(* Logix 5000 project; controller HP_SSC01hv vendor 1 type 14 code 158 rev 32.11; software revision 32.03; part 13 of 15 *)
(* tags used below, declared in another part *)
   A_C1_0200 : ALIAS FOR S_C1_FaultSafety.0;
   A_C1_0201 : ALIAS FOR S_C1_FaultSafety.1;
   A_C1_0202 : ALIAS FOR S_C1_FaultSafety.2;
   A_C1_0203 : ALIAS FOR S_C1_FaultSafety.3;
   A_C1_0204 : ALIAS FOR S_C1_FaultSafety.4;
   A_C1_0206 : ALIAS FOR S_C1_FaultSafety.6;
   A_C1_0208 : ALIAS FOR S_C1_FaultSafety.8;
   A_C1_0209 : ALIAS FOR S_C1_FaultSafety.9;
   A_C1_0210 : ALIAS FOR S_C1_FaultSafety.10;
   A_C1_0211 : ALIAS FOR S_C1_FaultSafety.11;
   A_C1_0216 : ALIAS FOR S_C1_FaultSafety.16;
   A_C1_0217 : ALIAS FOR S_C1_FaultSafety.17;
   A_C1_0220 : ALIAS FOR S_C1_FaultSafety.20;
   A_C2_0200 : ALIAS FOR S_C2_FaultSafety.0;
   A_C2_0201 : ALIAS FOR S_C2_FaultSafety.1;
   A_C2_0202 : ALIAS FOR S_C2_FaultSafety.2;
   A_C2_0203 : ALIAS FOR S_C2_FaultSafety.3;
   A_C2_0204 : ALIAS FOR S_C2_FaultSafety.4;
   A_C2_0206 : ALIAS FOR S_C2_FaultSafety.6;
   A_C2_0208 : ALIAS FOR S_C2_FaultSafety.8;
   A_C2_0209 : ALIAS FOR S_C2_FaultSafety.9;
   A_C2_0210 : ALIAS FOR S_C2_FaultSafety.10;
   A_C2_0211 : ALIAS FOR S_C2_FaultSafety.11;
   A_C2_0216 : ALIAS FOR S_C2_FaultSafety.16;
   A_C2_0217 : ALIAS FOR S_C2_FaultSafety.17;
   A_C2_0218 : ALIAS FOR S_C2_FaultSafety.18;
   A_C2_0219 : ALIAS FOR S_C2_FaultSafety.19;
   A_C2_0220 : ALIAS FOR S_C2_FaultSafety.20;
   A_C2_0221 : ALIAS FOR S_C2_FaultSafety.21;
   A_C2_0222 : ALIAS FOR S_C2_FaultSafety.22;
   A_C2_0223 : ALIAS FOR S_C2_FaultSafety.23;
   A_C2_0224 : ALIAS FOR S_C2_FaultSafety.24;
   A_C2_0230 : ALIAS FOR S_C2_FaultSafety.30;
   A_C2_0231 : ALIAS FOR S_C2_FaultSafety.31;
   A_S01_0104 : ALIAS FOR System_FaultSafeIO.4;
   A_S01_0122 : ALIAS FOR System_FaultSafeIO.22;
   C02_SafeMemory : Udt_Carsl_SafeData;
   C1_EvacInPositionTest : DINT;
   Multiplier : DINT;
   none : BOOL;
   RCS_CMD_EvacToStation : BOOL;
   RCS_SafeMemory_S01 : Udt_RCS_SafeData;
   RCS_SyncMotionEnable : BOOL;
   S1_C1_SafeOffFdbkRIN : REDUNDANT_INPUT;
   S_C1_AtEvacSpeed : BOOL;
   S_C1_BrakeTest : BOOL;
   S_C1_CircuitReset : BOOL;
   S_C1_CircuitReset_Pulse : TIMER;
   S_C1_DrawBridge_LS1 : ALIAS FOR SSC01_Safe2:I.Pt00Data;
   S_C1_DrawBridge_LS2 : ALIAS FOR SSC01_Safe2:I.Pt01Data;
   S_C1_DrawbridgeInputOK : BOOL;
   S_C1_DrawbridgeRIN : REDUNDANT_INPUT;
   S_C1_DumpTest : BOOL;
   S_C1_EvacOk : BOOL;
   S_C1_ExecuteInputOK : BOOL;
   S_C1_ExecutePB : BOOL;
   S_C1_FaultReset : BOOL;
   S_C1_FaultSafety : DINT;
   S_C1_FaultSafety_OK : BOOL;
   S_C1_FaultStandard : DINT;
   S_C1_FaultStandard_OK : BOOL;
   S_C1_FW_LocalOK : BOOL;
   S_C1_InEvacPosition : BOOL;
   S_C1_MaintEnable : BOOL;
   S_C1_MCC1_LIM_MCR : ALIAS FOR C1_Safe:O.Pt04Data;
   S_C1_ModeLocal : BOOL;
   S_C1_ModeRemote : BOOL;
   S_C1_MotionEnabled : BOOL;
   S_C1_MOTN_EXEC_RIN : REDUNDANT_INPUT;
   S_C1_MOTN_EXEC_SS_A : ALIAS FOR C1_Safe:I.Pt02Data;
   S_C1_MOTN_EXEC_SS_B : ALIAS FOR C1_Safe:I.Pt03Data;
   S_C1_MotorActualPositionX1000 : DINT;
   S_C1_MotorActualPositionX1000MOD60 : DINT;
   S_C1_MotorAverageVelocityX1000 : DINT;
   S_C1_MStop : EMERGENCY_STOP;
   S_C1_MSTOP_A : ALIAS FOR C1_Safe:I.Pt06Data;
   S_C1_MSTOP_B : ALIAS FOR C1_Safe:I.Pt07Data;
   S_C1_MSTOP_InputOK : BOOL;
   S_C1_MSTOP_LT : ALIAS FOR C1_Safe:O.Pt02Data;
   S_C1_NearOnPath : BOOL;
   S_C1_NearOnPathHi : DINT;
   S_C1_NearOnPathHiBase : DINT;
   S_C1_NearOnPathLow : DINT;
   S_C1_NearOnPathLowBase : DINT;
   S_C1_OffPath : BOOL;
   S_C1_OIT_FaultReset : BOOL;
   S_C1_OnPath : BOOL;
   S_C1_OnPathHi : DINT;
   S_C1_OnPathLow : DINT;
   S_C1_ONS : DINT;
   S_C1_ONS_CircuitFault : BOOL;
   S_C1_ONS_Status : BOOL;
   S_C1_OutputEnable : BOOL;
   S_C1_PathError : DINT;
   S_C1_PathErrorTest : DINT;
   S_C1_PathErrorTestTemp : DINT;
   S_C1_PathErrorTestTemp2 : DINT;
   S_C1_PathOffset : DINT;
   S_C1_PressureOK : ALIAS FOR C1_Safe:I.Pt05Data;
   S_C1_ResetTOF : TIMER;
   S_C1_SAFE_FDBK_Aux1 : BOOL;
   S_C1_SAFE_FDBK_Aux2 : BOOL;
   S_C1_SAFE_OFF_FDBK1 : ALIAS FOR C1_Safe:I.Pt01Data;
   S_C1_SAFE_OFF_FDBK2 : ALIAS FOR C1_Safe:I.Pt00Data;
   S_C1_SafeOff_ROUT : REDUNDANT_OUTPUT;
   S_C1_SafeOffEnabled : BOOL;
   S_C1_SafeOffEngaged : BOOL;
   S_C1_SafeOffInputOK : BOOL;
   S_C1_SAFETY_ENABLE_1 : ALIAS FOR C1_Safe:O.Pt00Data;
   S_C1_SAFETY_ENABLE_2 : ALIAS FOR C1_Safe:O.Pt01Data;
   S_C1_SS_RemoteMode : BOOL;
   S_C1_Stop0_OK : BOOL;
   S_C1_Stop1_OK : BOOL;
   S_C1_Stop1_OK_TOF : TIMER;
   S_C1_WindowAdderTemp1 : DINT;
   S_C1_WindowAdderTemp2 : DINT;
   S_C1_WindowAdderTemp3 : DINT;
   S_C2_AtEvacSpeed : BOOL;
   S_C2_BrakeRelease : ALIAS FOR C2_Safe:O.Pt06Data;
   S_C2_BrakeReleaseSelected : BOOL;
   S_C2_BrakeTest : BOOL;
   S_C2_CircuitReset : BOOL;
   S_C2_DrawbridgeInputOK : BOOL;
   S_C2_DrawbridgeRIN : REDUNDANT_INPUT;
   S_C2_DumpValveRelease : ALIAS FOR C2_Safe:O.Pt05Data;
   S_C2_DumpValveReleaseSelected : BOOL;
   S_C2_EncoderBuffer : DINT[4];
   S_C2_EncoderChange : DINT;
   S_C2_EncoderCounter : DINT;
   S_C2_EncoderCounts : DINT;
   S_C2_EncoderPositionAtHome : DINT;
   S_C2_EncoderPositionAtHomeSet : BOOL;
   S_C2_EncoderPositionDegree : DINT;
   S_C2_EncoderRev : DINT;
   S_C2_EncoderRevX1000 : DINT;
   S_C2_EncoderTemp : DINT;
   S_C2_EncoderTemp2 : DINT;
   S_C2_EvacOK : BOOL;
   S_C2_ExecuteInputOK : BOOL;
   S_C2_FaultReset : BOOL;
   S_C2_FaultSafety : DINT;
   S_C2_FaultSafety_OK : BOOL;
   S_C2_FaultStandard_OK : BOOL;
   S_C2_FaultTimer : TIMER[8];
   S_C2_Homed : BOOL;
   S_C2_HomeInputStatus : BOOL;
   S_C2_HomeSafePE : ALIAS FOR C2_Safe:I.Pt04Data;
   S_C2_InEvacPosition : BOOL;
   S_C2_ModeLocal : BOOL;
   S_C2_ModeRemote : BOOL;
   S_C2_MotorActualPositionX1000 : DINT;
   S_C2_MotorActualPositionX1000MOD60 : DINT;
   S_C2_MotorAverageVelocityX1000 : DINT;
   S_C2_MotorToEncoderError : DINT;
   S_C2_MStop : EMERGENCY_STOP;
   S_C2_MSTOP_InputOK : BOOL;
   S_C2_NearOnPath : BOOL;
   S_C2_NearOnPathHi : DINT;
   S_C2_NearOnPathHiBase : DINT;
   S_C2_NearOnPathLow : DINT;
   S_C2_NearOnPathLowBase : DINT;
   S_C2_OffPath : BOOL;
   S_C2_OnPath : BOOL;
   S_C2_OnPathHi : DINT;
   S_C2_OnPathLow : DINT;
   S_C2_ONS_Fault : BOOL;
   S_C2_OutputEnable : BOOL;
   S_C2_PathError : DINT;
   S_C2_PathErrorTest : DINT;
   S_C2_PathErrorTestTemp : DINT;
   S_C2_PathErrorTestTemp2 : DINT;
   S_C2_PathOffset : DINT;
   S_C2_PressureOK : ALIAS FOR C2_Safe:I.Pt05Data;
   S_C2_RemoteBrakeAndHomeSequence : DINT;
   S_C2_ReverseMotionDebounce : TIMER;
   S_C2_SAFE_OFF_FDBK1 : ALIAS FOR C2_Safe:I.Pt01Data;
   S_C2_SAFE_OFF_FDBK2 : ALIAS FOR C2_Safe:I.Pt00Data;
   S_C2_SafeOff_ROUT : REDUNDANT_OUTPUT;
   S_C2_SafeOffInputOK : BOOL;
   S_C2_SetEncoderHomePosition : BOOL;
   S_C2_WindowAdderTemp1 : DINT;
   S_C2_WindowAdderTemp2 : DINT;
   S_C2_WindowAdderTemp3 : DINT;
   S_EncoderRollover : DINT;
   S_EvacToStationTON : TIMER;
   S_FlashOn : TIMER;
   S_RCS_CMD_FaultReset : BOOL;
   S_RCS_EvacSpeedStart_TON : TIMER;
   S_RCS_MasterPositionDegrees : DINT;
   S_RCS_MotionEnable : BOOL;
   S_System_FaultStandard : DINT;
   SSC_Rail_BypassOK : BOOL;
   SSC_SafeFlt_OK : BOOL;
   SSC_SafetyIO_OK : BOOL;
   SSC_StdFlt_OK : BOOL;
   SSC_Stop0_OK : BOOL;
   SSC_Stop1_OK : BOOL;
(* SafeCarousel1, continued *)

ROUTINE SC125_PathError   (* ladder *)
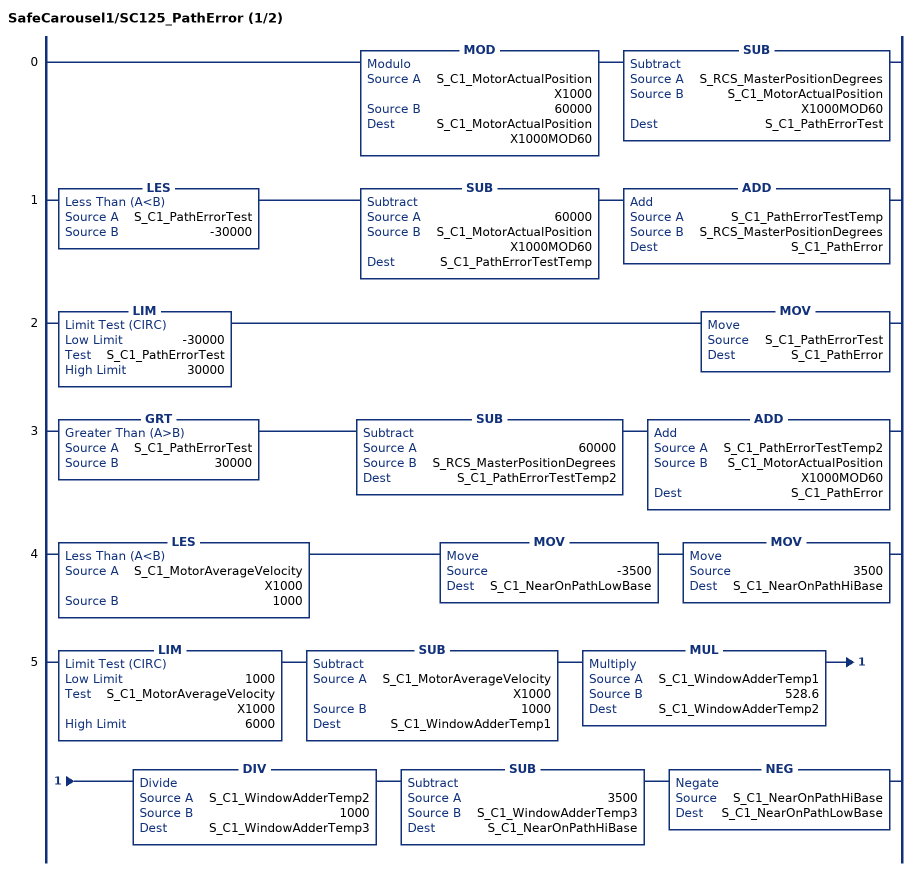
   0: MOD(S_C1_MotorActualPositionX1000,60000,S_C1_MotorActualPositionX1000MOD60)SUB(S_RCS_MasterPositionDegrees,S_C1_MotorActualPositionX1000MOD60,S_C1_PathErrorTest);
   1: LES(S_C1_PathErrorTest,-30000)SUB(60000,S_C1_MotorActualPositionX1000MOD60,S_C1_PathErrorTestTemp)ADD(S_C1_PathErrorTestTemp,S_RCS_MasterPositionDegrees,S_C1_PathError);
   2: LIM(-30000,S_C1_PathErrorTest,30000)MOV(S_C1_PathErrorTest,S_C1_PathError);
   3: GRT(S_C1_PathErrorTest,30000)SUB(60000,S_RCS_MasterPositionDegrees,S_C1_PathErrorTestTemp2)ADD(S_C1_PathErrorTestTemp2,S_C1_MotorActualPositionX1000MOD60,S_C1_PathError);
   4: LES(S_C1_MotorAverageVelocityX1000,1000)MOV(-3500,S_C1_NearOnPathLowBase)MOV(3500,S_C1_NearOnPathHiBase);
   5: LIM(1000,S_C1_MotorAverageVelocityX1000,6000)SUB(S_C1_MotorAverageVelocityX1000,1000,S_C1_WindowAdderTemp1)MUL(S_C1_WindowAdderTemp1,528.6,S_C1_WindowAdderTemp2)DIV(S_C1_WindowAdderTemp2,1000,S_C1_WindowAdderTemp3)SUB(3500,S_C1_WindowAdderTemp3,S_C1_NearOnPathHiBase)NEG(S_C1_NearOnPathHiBase,S_C1_NearOnPathLowBase);
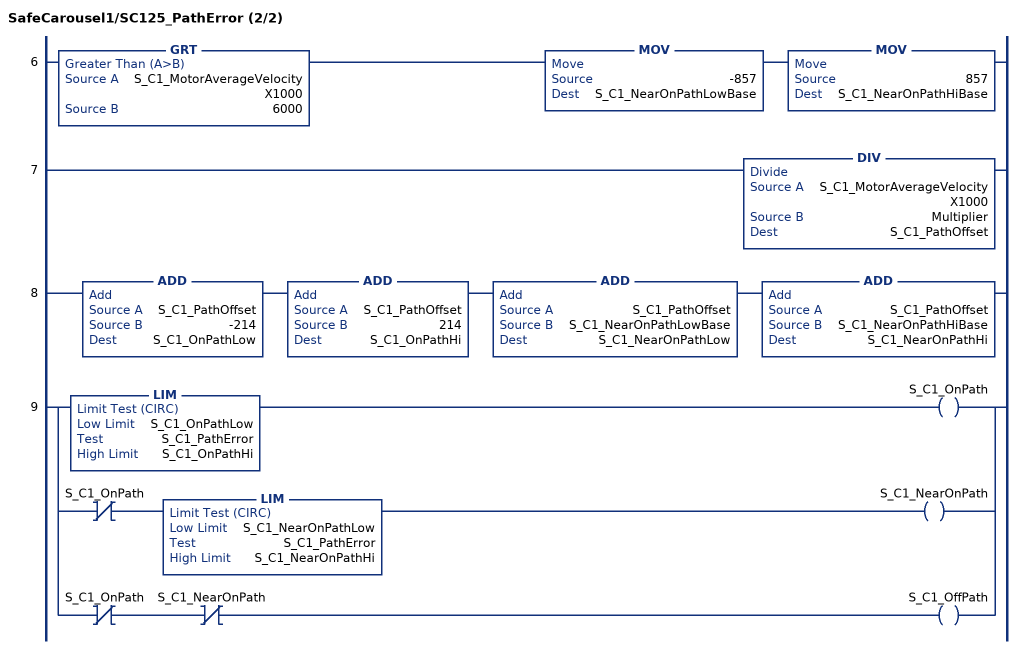
   6: GRT(S_C1_MotorAverageVelocityX1000,6000)MOV(-857,S_C1_NearOnPathLowBase)MOV(857,S_C1_NearOnPathHiBase);
   7: DIV(S_C1_MotorAverageVelocityX1000,Multiplier,S_C1_PathOffset);
   8: ADD(S_C1_PathOffset,-214,S_C1_OnPathLow)ADD(S_C1_PathOffset,214,S_C1_OnPathHi)ADD(S_C1_PathOffset,S_C1_NearOnPathLowBase,S_C1_NearOnPathLow)ADD(S_C1_PathOffset,S_C1_NearOnPathHiBase,S_C1_NearOnPathHi);
   9: [LIM(S_C1_OnPathLow,S_C1_PathError,S_C1_OnPathHi) OTE(S_C1_OnPath) ,XIO(S_C1_OnPath) LIM(S_C1_NearOnPathLow,S_C1_PathError,S_C1_NearOnPathHi) OTE(S_C1_NearOnPath) ,XIO(S_C1_OnPath) XIO(S_C1_NearOnPath) OTE(S_C1_OffPath) ];
END_ROUTINE

ROUTINE SC130_SafetyInputs   (* ladder *)
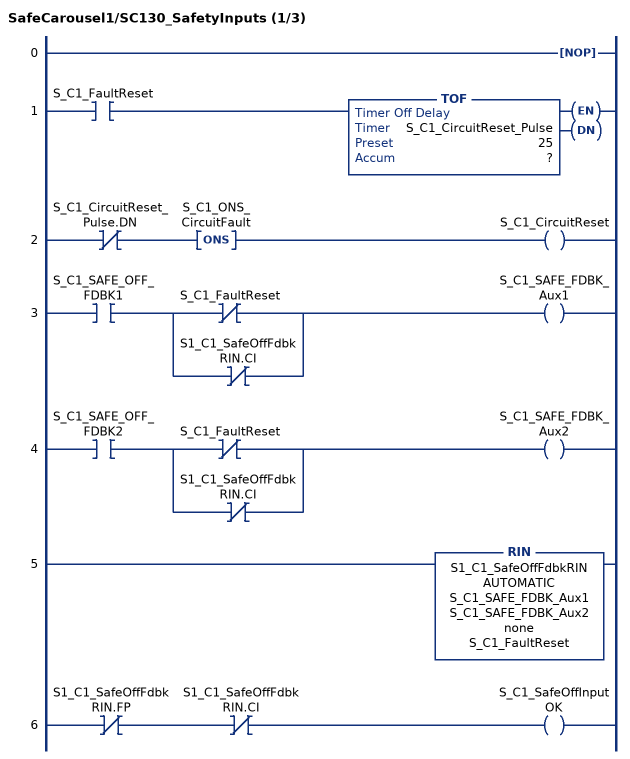
   0: NOP();
   1: XIC(S_C1_FaultReset)TOF(S_C1_CircuitReset_Pulse,?,?);
   2: XIO(S_C1_CircuitReset_Pulse.DN)ONS(S_C1_ONS_CircuitFault)OTE(S_C1_CircuitReset);
   3: XIC(S_C1_SAFE_OFF_FDBK1)[XIO(S_C1_FaultReset) ,XIO(S1_C1_SafeOffFdbkRIN.CI) ]OTE(S_C1_SAFE_FDBK_Aux1);
   4: XIC(S_C1_SAFE_OFF_FDBK2)[XIO(S_C1_FaultReset) ,XIO(S1_C1_SafeOffFdbkRIN.CI) ]OTE(S_C1_SAFE_FDBK_Aux2);
   5: RIN(S1_C1_SafeOffFdbkRIN,AUTOMATIC,S_C1_SAFE_FDBK_Aux1,S_C1_SAFE_FDBK_Aux2,none,S_C1_FaultReset);
   6: XIO(S1_C1_SafeOffFdbkRIN.FP)XIO(S1_C1_SafeOffFdbkRIN.CI)OTE(S_C1_SafeOffInputOK);
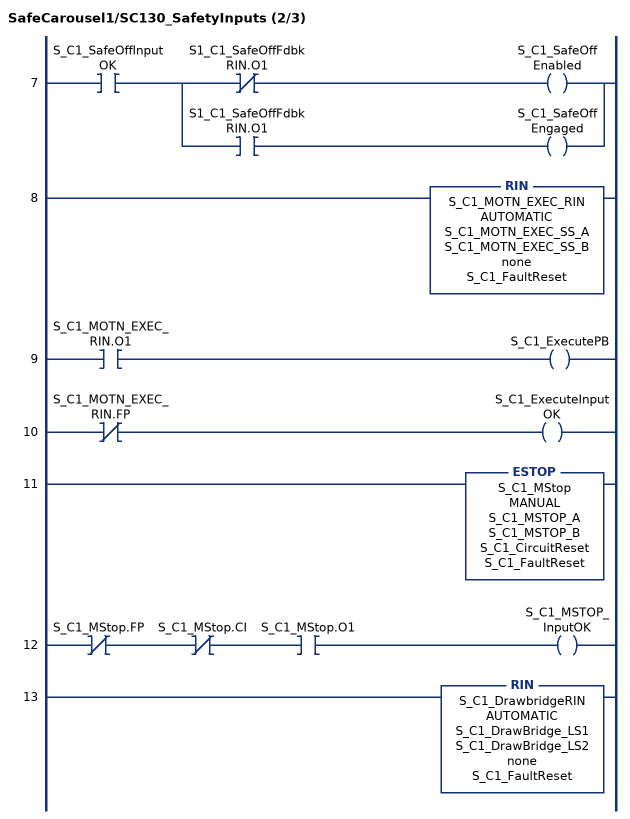
   7: XIC(S_C1_SafeOffInputOK)[XIO(S1_C1_SafeOffFdbkRIN.O1) OTE(S_C1_SafeOffEnabled) ,XIC(S1_C1_SafeOffFdbkRIN.O1) OTE(S_C1_SafeOffEngaged) ];
   8: RIN(S_C1_MOTN_EXEC_RIN,AUTOMATIC,S_C1_MOTN_EXEC_SS_A,S_C1_MOTN_EXEC_SS_B,none,S_C1_FaultReset);
   9: XIC(S_C1_MOTN_EXEC_RIN.O1)OTE(S_C1_ExecutePB);
   10: XIO(S_C1_MOTN_EXEC_RIN.FP)OTE(S_C1_ExecuteInputOK);
   11: ESTOP(S_C1_MStop,MANUAL,S_C1_MSTOP_A,S_C1_MSTOP_B,S_C1_CircuitReset,S_C1_FaultReset);
   12: XIO(S_C1_MStop.FP)XIO(S_C1_MStop.CI)XIC(S_C1_MStop.O1)OTE(S_C1_MSTOP_InputOK);
   13: RIN(S_C1_DrawbridgeRIN,AUTOMATIC,S_C1_DrawBridge_LS1,S_C1_DrawBridge_LS2,none,S_C1_FaultReset);
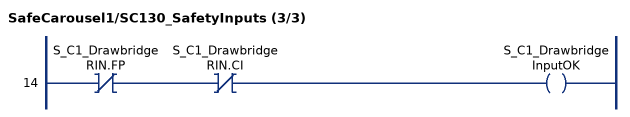
   14: XIO(S_C1_DrawbridgeRIN.FP)XIO(S_C1_DrawbridgeRIN.CI)OTE(S_C1_DrawbridgeInputOK);
END_ROUTINE

ROUTINE SC135_SafetyOutputs   (* ladder *)
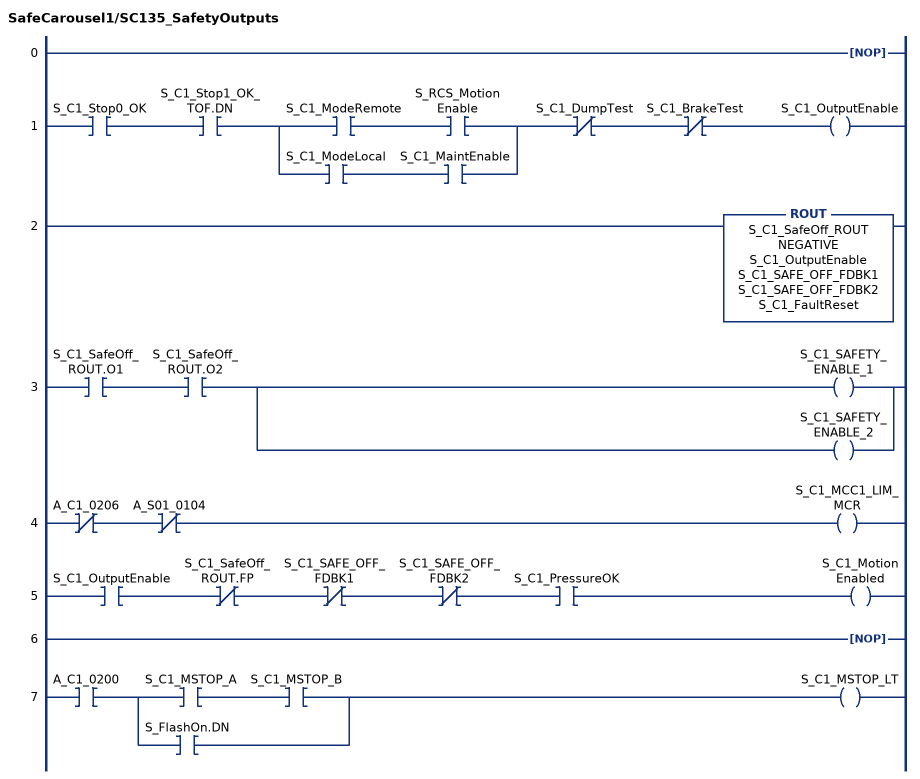
   0: NOP();
   1: XIC(S_C1_Stop0_OK)XIC(S_C1_Stop1_OK_TOF.DN)[XIC(S_C1_ModeRemote) XIC(S_RCS_MotionEnable) ,XIC(S_C1_ModeLocal) XIC(S_C1_MaintEnable) ]XIO(S_C1_DumpTest)XIO(S_C1_BrakeTest)OTE(S_C1_OutputEnable);
   2: ROUT(S_C1_SafeOff_ROUT,NEGATIVE,S_C1_OutputEnable,S_C1_SAFE_OFF_FDBK1,S_C1_SAFE_OFF_FDBK2,S_C1_FaultReset);
   3: XIC(S_C1_SafeOff_ROUT.O1)XIC(S_C1_SafeOff_ROUT.O2)[OTE(S_C1_SAFETY_ENABLE_1) ,OTE(S_C1_SAFETY_ENABLE_2) ];
   4: XIO(A_C1_0206)XIO(A_S01_0104)OTE(S_C1_MCC1_LIM_MCR);
   5: XIC(S_C1_OutputEnable)XIO(S_C1_SafeOff_ROUT.FP)XIO(S_C1_SAFE_OFF_FDBK1)XIO(S_C1_SAFE_OFF_FDBK2)XIC(S_C1_PressureOK)OTE(S_C1_MotionEnabled);
   6: NOP();
   7: XIC(A_C1_0200)[XIC(S_C1_MSTOP_A) XIC(S_C1_MSTOP_B) ,XIC(S_FlashOn.DN) ]OTE(S_C1_MSTOP_LT);
END_ROUTINE

ROUTINE SC140_Status   (* ladder *)
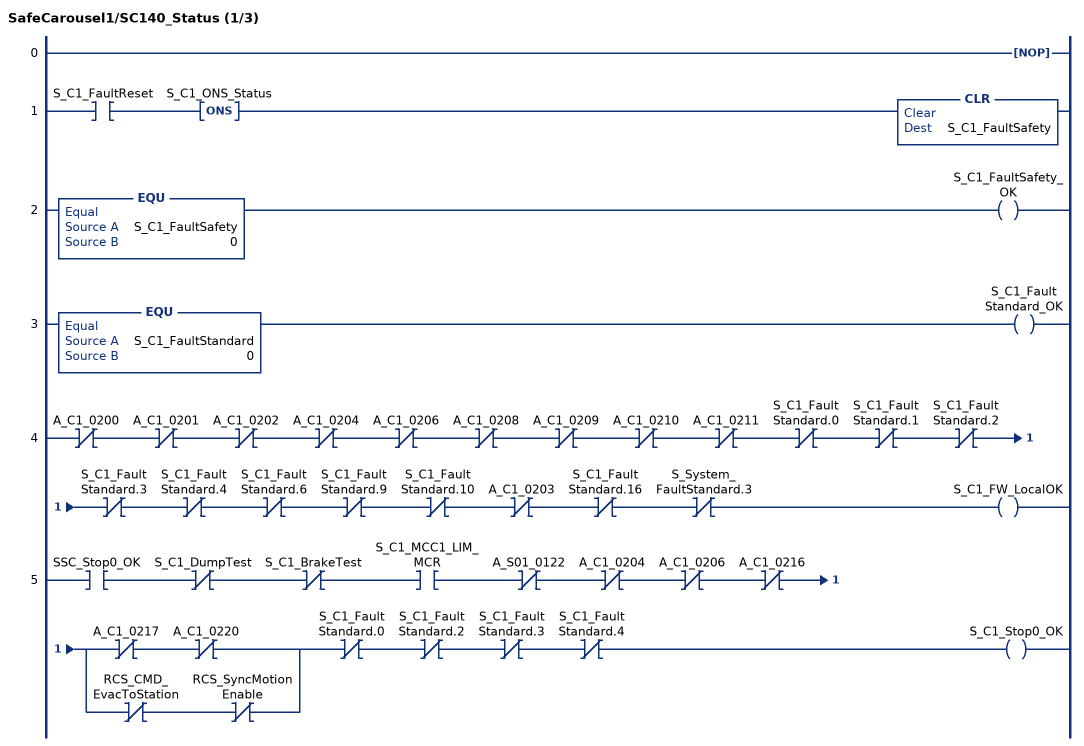
   0: NOP();
   1: XIC(S_C1_FaultReset)ONS(S_C1_ONS_Status)CLR(S_C1_FaultSafety);
   2: EQU(S_C1_FaultSafety,0)OTE(S_C1_FaultSafety_OK);
   3: EQU(S_C1_FaultStandard,0)OTE(S_C1_FaultStandard_OK);
   4: XIO(A_C1_0200)XIO(A_C1_0201)XIO(A_C1_0202)XIO(A_C1_0204)XIO(A_C1_0206)XIO(A_C1_0208)XIO(A_C1_0209)XIO(A_C1_0210)XIO(A_C1_0211)XIO(S_C1_FaultStandard.0)XIO(S_C1_FaultStandard.1)XIO(S_C1_FaultStandard.2)XIO(S_C1_FaultStandard.3)XIO(S_C1_FaultStandard.4)XIO(S_C1_FaultStandard.6)XIO(S_C1_FaultStandard.9)XIO(S_C1_FaultStandard.10)XIO(A_C1_0203)XIO(S_C1_FaultStandard.16)XIO(S_System_FaultStandard.3)OTE(S_C1_FW_LocalOK);
   5: XIC(SSC_Stop0_OK)XIO(S_C1_DumpTest)XIO(S_C1_BrakeTest)XIC(S_C1_MCC1_LIM_MCR)XIO(A_S01_0122)XIO(A_C1_0204)XIO(A_C1_0206)XIO(A_C1_0216)[XIO(A_C1_0217) XIO(A_C1_0220) ,XIO(RCS_CMD_EvacToStation) XIO(RCS_SyncMotionEnable) ]XIO(S_C1_FaultStandard.0)XIO(S_C1_FaultStandard.2)XIO(S_C1_FaultStandard.3)XIO(S_C1_FaultStandard.4)OTE(S_C1_Stop0_OK);
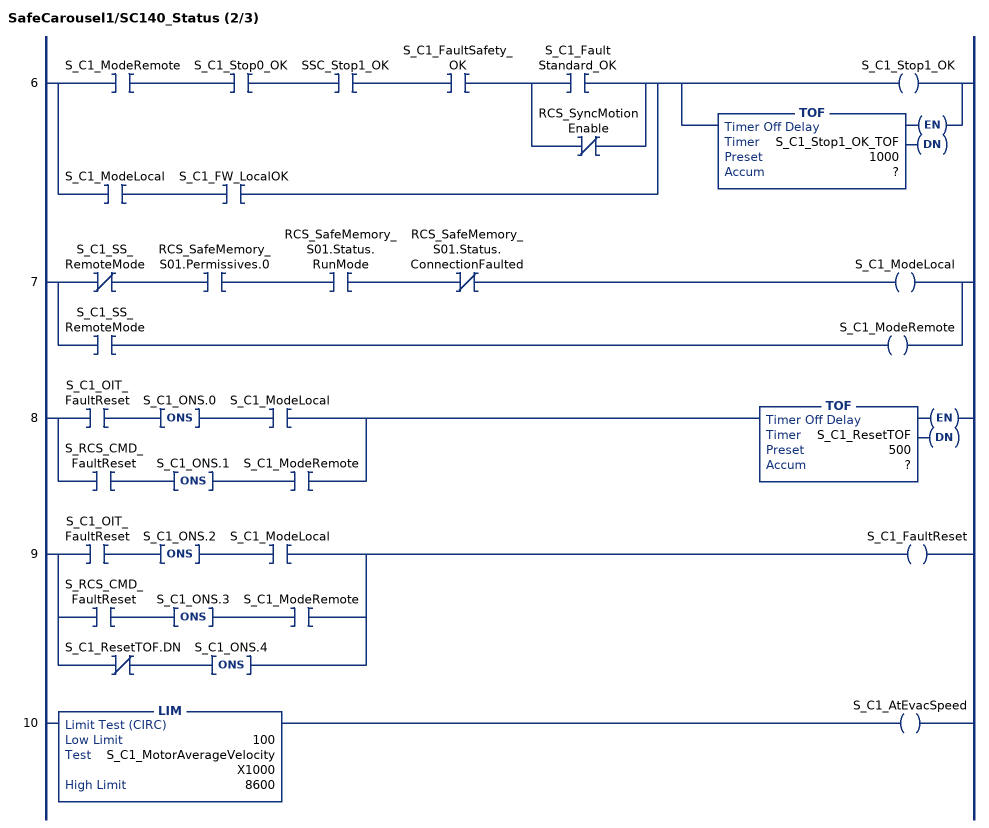
   6: [XIC(S_C1_ModeRemote) XIC(S_C1_Stop0_OK) XIC(SSC_Stop1_OK) XIC(S_C1_FaultSafety_OK) [XIC(S_C1_FaultStandard_OK) ,XIO(RCS_SyncMotionEnable) ] ,XIC(S_C1_ModeLocal) XIC(S_C1_FW_LocalOK) ][OTE(S_C1_Stop1_OK) ,TOF(S_C1_Stop1_OK_TOF,?,?) ];
   7: [XIO(S_C1_SS_RemoteMode) XIC(RCS_SafeMemory_S01.Permissives.0) XIC(RCS_SafeMemory_S01.Status.RunMode) XIO(RCS_SafeMemory_S01.Status.ConnectionFaulted) OTE(S_C1_ModeLocal) ,XIC(S_C1_SS_RemoteMode) OTE(S_C1_ModeRemote) ];
   8: [XIC(S_C1_OIT_FaultReset) ONS(S_C1_ONS.0) XIC(S_C1_ModeLocal) ,XIC(S_RCS_CMD_FaultReset) ONS(S_C1_ONS.1) XIC(S_C1_ModeRemote) ]TOF(S_C1_ResetTOF,?,?);
   9: [XIC(S_C1_OIT_FaultReset) ONS(S_C1_ONS.2) XIC(S_C1_ModeLocal) ,XIC(S_RCS_CMD_FaultReset) ONS(S_C1_ONS.3) XIC(S_C1_ModeRemote) ,XIO(S_C1_ResetTOF.DN) ONS(S_C1_ONS.4) ]OTE(S_C1_FaultReset);
   10: LIM(100,S_C1_MotorAverageVelocityX1000,8600)OTE(S_C1_AtEvacSpeed);
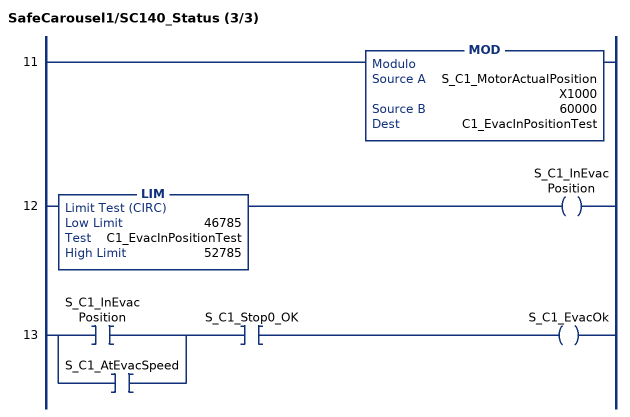
   11: MOD(S_C1_MotorActualPositionX1000,60000,C1_EvacInPositionTest);
   12: LIM(46785,C1_EvacInPositionTest,52785)OTE(S_C1_InEvacPosition);
   13: [XIC(S_C1_InEvacPosition) ,XIC(S_C1_AtEvacSpeed) ]XIC(S_C1_Stop0_OK)OTE(S_C1_EvacOk);
END_ROUTINE
END_PROGRAM

PROGRAM SafeCarousel2   (* main routine SC200_Main, safety *)

ROUTINE SC200_Main   (* ladder *)
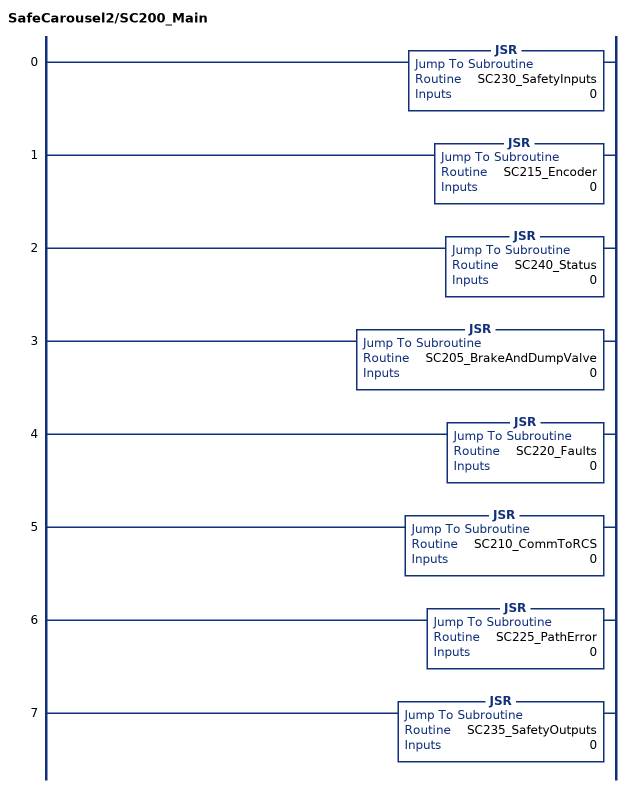
   0: JSR(SC230_SafetyInputs,0);
   1: JSR(SC215_Encoder,0);
   2: JSR(SC240_Status,0);
   3: JSR(SC205_BrakeAndDumpValve,0);
   4: JSR(SC220_Faults,0);
   5: JSR(SC210_CommToRCS,0);
   6: JSR(SC225_PathError,0);
   7: JSR(SC235_SafetyOutputs,0);
END_ROUTINE

ROUTINE SC205_BrakeAndDumpValve   (* ladder *)
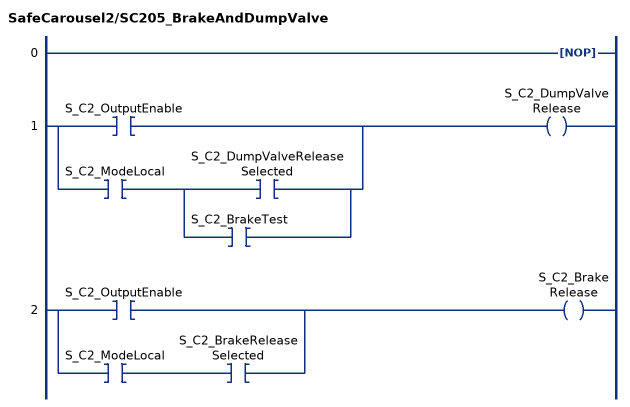
   0: NOP();
   1: [XIC(S_C2_OutputEnable) ,XIC(S_C2_ModeLocal) [XIC(S_C2_DumpValveReleaseSelected) ,XIC(S_C2_BrakeTest) ] ]OTE(S_C2_DumpValveRelease);
   2: [XIC(S_C2_OutputEnable) ,XIC(S_C2_ModeLocal) XIC(S_C2_BrakeReleaseSelected) ]OTE(S_C2_BrakeRelease);
END_ROUTINE

ROUTINE SC210_CommToRCS   (* ladder *)
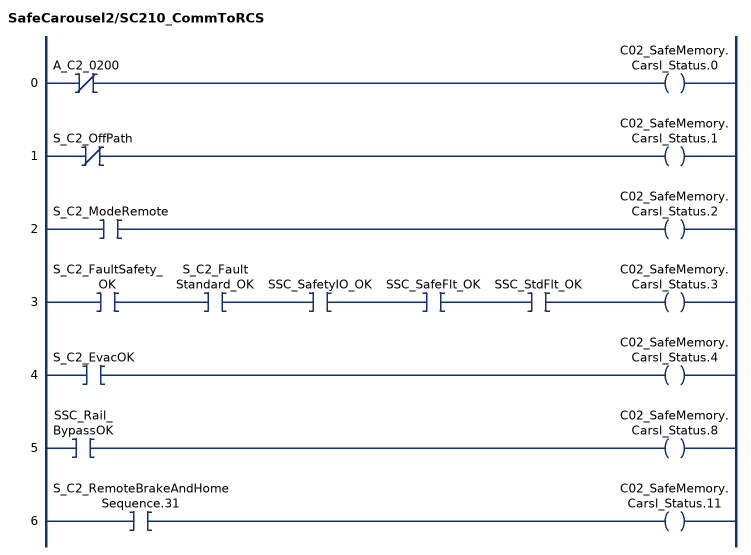
   0: XIO(A_C2_0200)OTE(C02_SafeMemory.Carsl_Status.0);
   1: XIO(S_C2_OffPath)OTE(C02_SafeMemory.Carsl_Status.1);
   2: XIC(S_C2_ModeRemote)OTE(C02_SafeMemory.Carsl_Status.2);
   3: XIC(S_C2_FaultSafety_OK)XIC(S_C2_FaultStandard_OK)XIC(SSC_SafetyIO_OK)XIC(SSC_SafeFlt_OK)XIC(SSC_StdFlt_OK)OTE(C02_SafeMemory.Carsl_Status.3);
   4: XIC(S_C2_EvacOK)OTE(C02_SafeMemory.Carsl_Status.4);
   5: XIC(SSC_Rail_BypassOK)OTE(C02_SafeMemory.Carsl_Status.8);
   6: XIC(S_C2_RemoteBrakeAndHomeSequence.31)OTE(C02_SafeMemory.Carsl_Status.11);
END_ROUTINE

ROUTINE SC215_Encoder   (* ladder *)
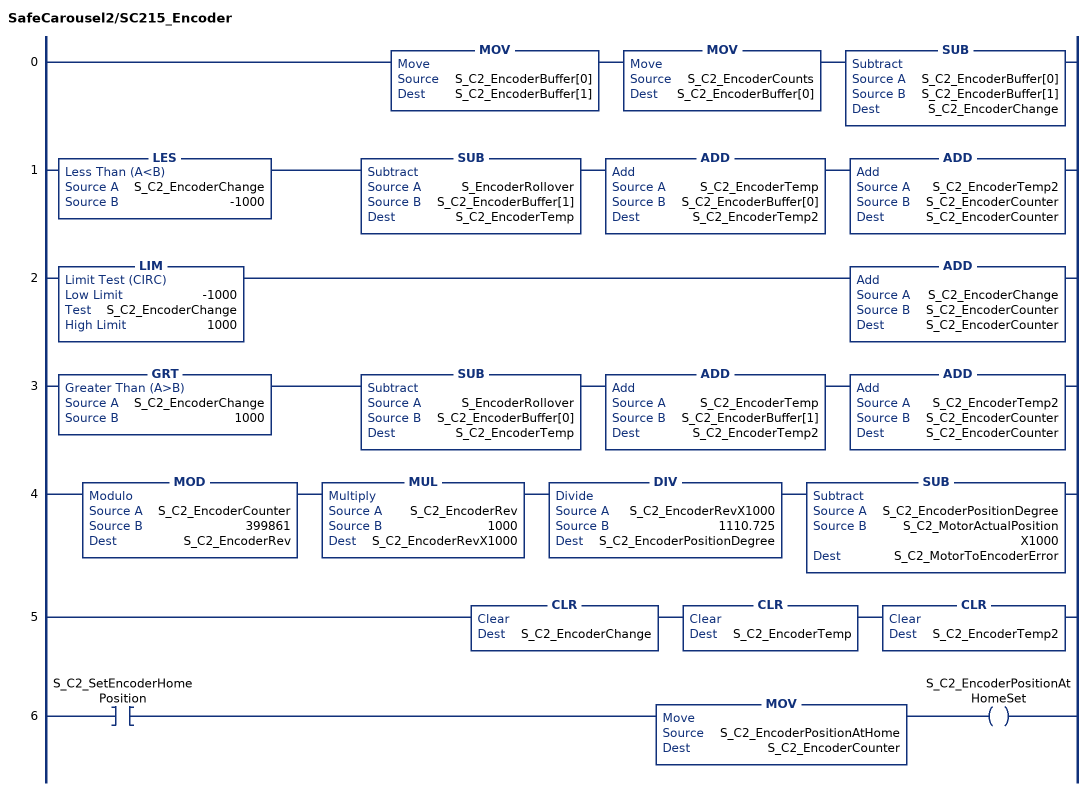
   0: MOV(S_C2_EncoderBuffer[0],S_C2_EncoderBuffer[1])MOV(S_C2_EncoderCounts,S_C2_EncoderBuffer[0])SUB(S_C2_EncoderBuffer[0],S_C2_EncoderBuffer[1],S_C2_EncoderChange);
   1: LES(S_C2_EncoderChange,-1000)SUB(S_EncoderRollover,S_C2_EncoderBuffer[1],S_C2_EncoderTemp)ADD(S_C2_EncoderTemp,S_C2_EncoderBuffer[0],S_C2_EncoderTemp2)ADD(S_C2_EncoderTemp2,S_C2_EncoderCounter,S_C2_EncoderCounter);
   2: LIM(-1000,S_C2_EncoderChange,1000)ADD(S_C2_EncoderChange,S_C2_EncoderCounter,S_C2_EncoderCounter);
   3: GRT(S_C2_EncoderChange,1000)SUB(S_EncoderRollover,S_C2_EncoderBuffer[0],S_C2_EncoderTemp)ADD(S_C2_EncoderTemp,S_C2_EncoderBuffer[1],S_C2_EncoderTemp2)ADD(S_C2_EncoderTemp2,S_C2_EncoderCounter,S_C2_EncoderCounter);
   4: MOD(S_C2_EncoderCounter,399861,S_C2_EncoderRev)MUL(S_C2_EncoderRev,1000,S_C2_EncoderRevX1000)DIV(S_C2_EncoderRevX1000,1110.725,S_C2_EncoderPositionDegree)SUB(S_C2_EncoderPositionDegree,S_C2_MotorActualPositionX1000,S_C2_MotorToEncoderError);
   5: CLR(S_C2_EncoderChange)CLR(S_C2_EncoderTemp)CLR(S_C2_EncoderTemp2);
   6: XIC(S_C2_SetEncoderHomePosition)MOV(S_C2_EncoderPositionAtHome,S_C2_EncoderCounter)OTE(S_C2_EncoderPositionAtHomeSet);
END_ROUTINE

ROUTINE SC220_Faults   (* ladder *)
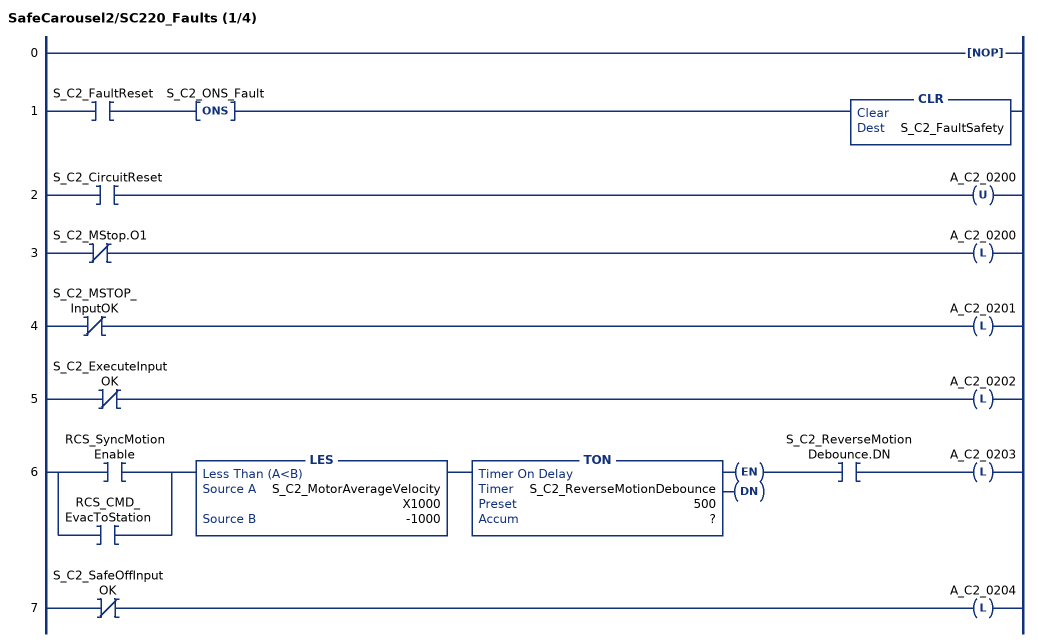
   0: NOP();
   1: XIC(S_C2_FaultReset)ONS(S_C2_ONS_Fault)CLR(S_C2_FaultSafety);
   2: XIC(S_C2_CircuitReset)OTU(A_C2_0200);
   3: XIO(S_C2_MStop.O1)OTL(A_C2_0200);
   4: XIO(S_C2_MSTOP_InputOK)OTL(A_C2_0201);
   5: XIO(S_C2_ExecuteInputOK)OTL(A_C2_0202);
   6: [XIC(RCS_SyncMotionEnable) ,XIC(RCS_CMD_EvacToStation) ]LES(S_C2_MotorAverageVelocityX1000,-1000)TON(S_C2_ReverseMotionDebounce,?,?)XIC(S_C2_ReverseMotionDebounce.DN)OTL(A_C2_0203);
   7: XIO(S_C2_SafeOffInputOK)OTL(A_C2_0204);
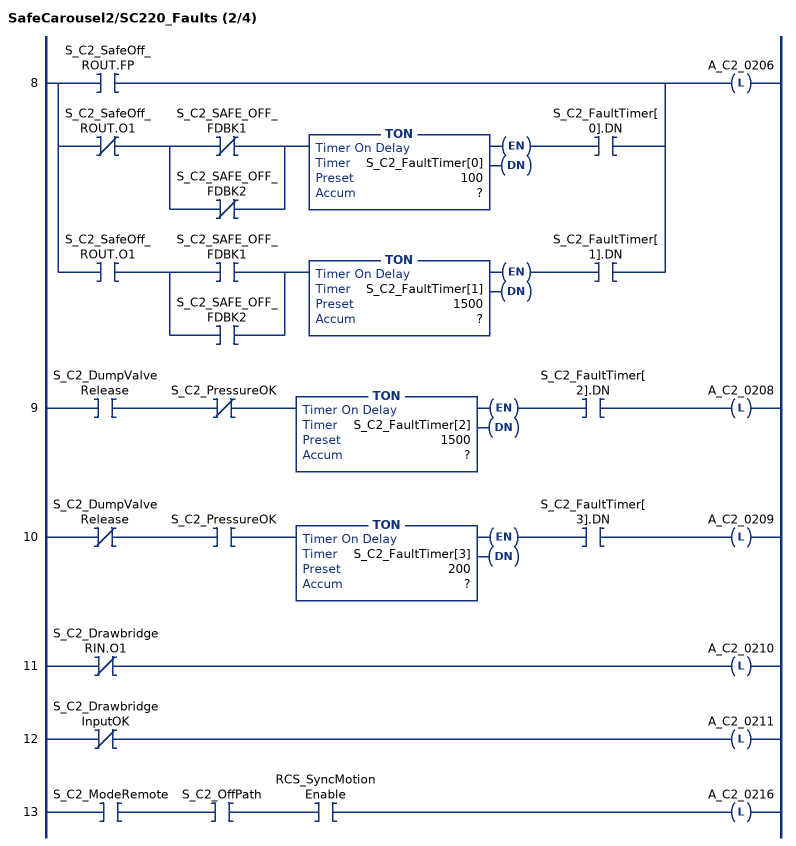
   8: [XIC(S_C2_SafeOff_ROUT.FP) ,XIO(S_C2_SafeOff_ROUT.O1) [XIO(S_C2_SAFE_OFF_FDBK1) ,XIO(S_C2_SAFE_OFF_FDBK2) ] TON(S_C2_FaultTimer[0],?,?) XIC(S_C2_FaultTimer[0].DN) ,XIC(S_C2_SafeOff_ROUT.O1) [XIC(S_C2_SAFE_OFF_FDBK1) ,XIC(S_C2_SAFE_OFF_FDBK2) ] TON(S_C2_FaultTimer[1],?,?) XIC(S_C2_FaultTimer[1].DN) ]OTL(A_C2_0206);
   9: XIC(S_C2_DumpValveRelease)XIO(S_C2_PressureOK)TON(S_C2_FaultTimer[2],?,?)XIC(S_C2_FaultTimer[2].DN)OTL(A_C2_0208);
   10: XIO(S_C2_DumpValveRelease)XIC(S_C2_PressureOK)TON(S_C2_FaultTimer[3],?,?)XIC(S_C2_FaultTimer[3].DN)OTL(A_C2_0209);
   11: XIO(S_C2_DrawbridgeRIN.O1)OTL(A_C2_0210);
   12: XIO(S_C2_DrawbridgeInputOK)OTL(A_C2_0211);
   13: XIC(S_C2_ModeRemote)XIC(S_C2_OffPath)XIC(RCS_SyncMotionEnable)OTL(A_C2_0216);
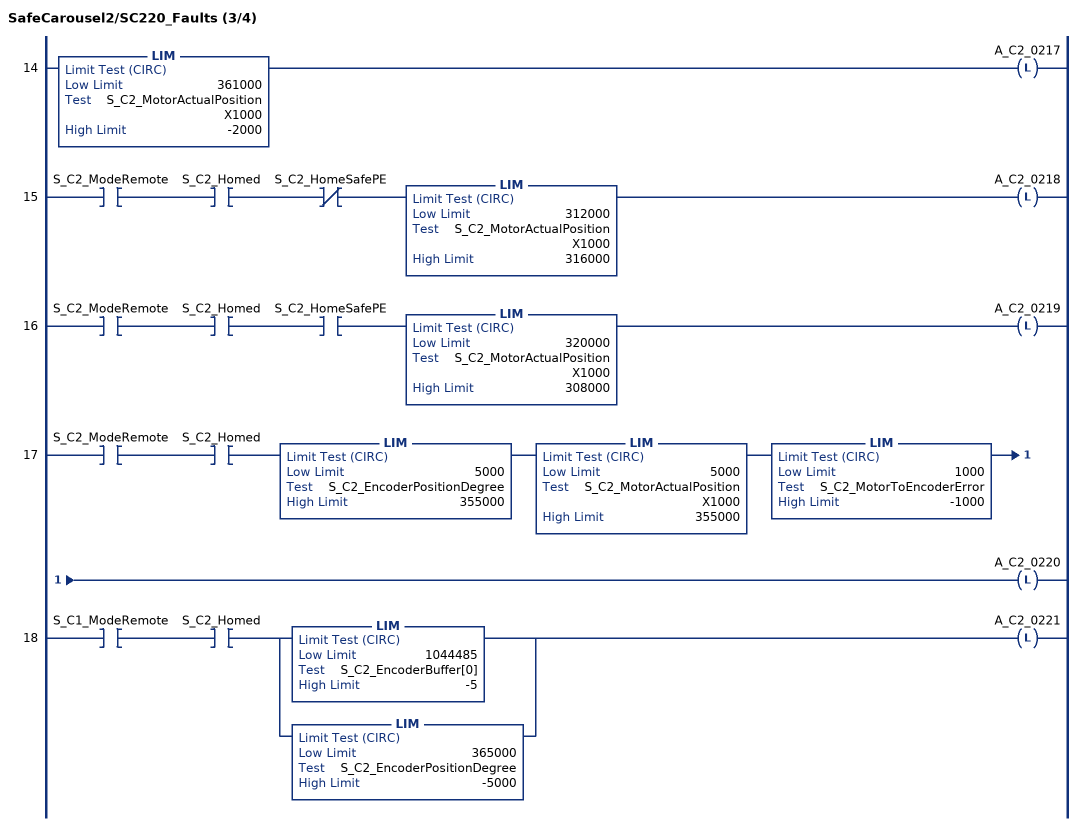
   14: LIM(361000,S_C2_MotorActualPositionX1000,-2000)OTL(A_C2_0217);
   15: XIC(S_C2_ModeRemote)XIC(S_C2_Homed)XIO(S_C2_HomeSafePE)LIM(312000,S_C2_MotorActualPositionX1000,316000)OTL(A_C2_0218);
   16: XIC(S_C2_ModeRemote)XIC(S_C2_Homed)XIC(S_C2_HomeSafePE)LIM(320000,S_C2_MotorActualPositionX1000,308000)OTL(A_C2_0219);
   17: XIC(S_C2_ModeRemote)XIC(S_C2_Homed)LIM(5000,S_C2_EncoderPositionDegree,355000)LIM(5000,S_C2_MotorActualPositionX1000,355000)LIM(1000,S_C2_MotorToEncoderError,-1000)OTL(A_C2_0220);
   18: XIC(S_C1_ModeRemote)XIC(S_C2_Homed)[LIM(1044485,S_C2_EncoderBuffer[0],-5) ,LIM(365000,S_C2_EncoderPositionDegree,-5000) ]OTL(A_C2_0221);
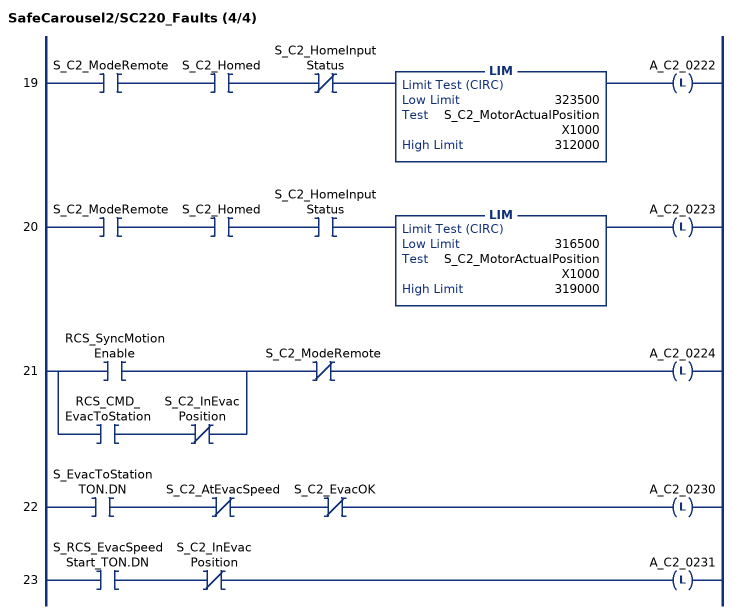
   19: XIC(S_C2_ModeRemote)XIC(S_C2_Homed)XIO(S_C2_HomeInputStatus)LIM(323500,S_C2_MotorActualPositionX1000,312000)OTL(A_C2_0222);
   20: XIC(S_C2_ModeRemote)XIC(S_C2_Homed)XIC(S_C2_HomeInputStatus)LIM(316500,S_C2_MotorActualPositionX1000,319000)OTL(A_C2_0223);
   21: [XIC(RCS_SyncMotionEnable) ,XIC(RCS_CMD_EvacToStation) XIO(S_C2_InEvacPosition) ]XIO(S_C2_ModeRemote)OTL(A_C2_0224);
   22: XIC(S_EvacToStationTON.DN)XIO(S_C2_AtEvacSpeed)XIO(S_C2_EvacOK)OTL(A_C2_0230);
   23: XIC(S_RCS_EvacSpeedStart_TON.DN)XIO(S_C2_InEvacPosition)OTL(A_C2_0231);
END_ROUTINE

ROUTINE SC225_PathError   (* ladder *)
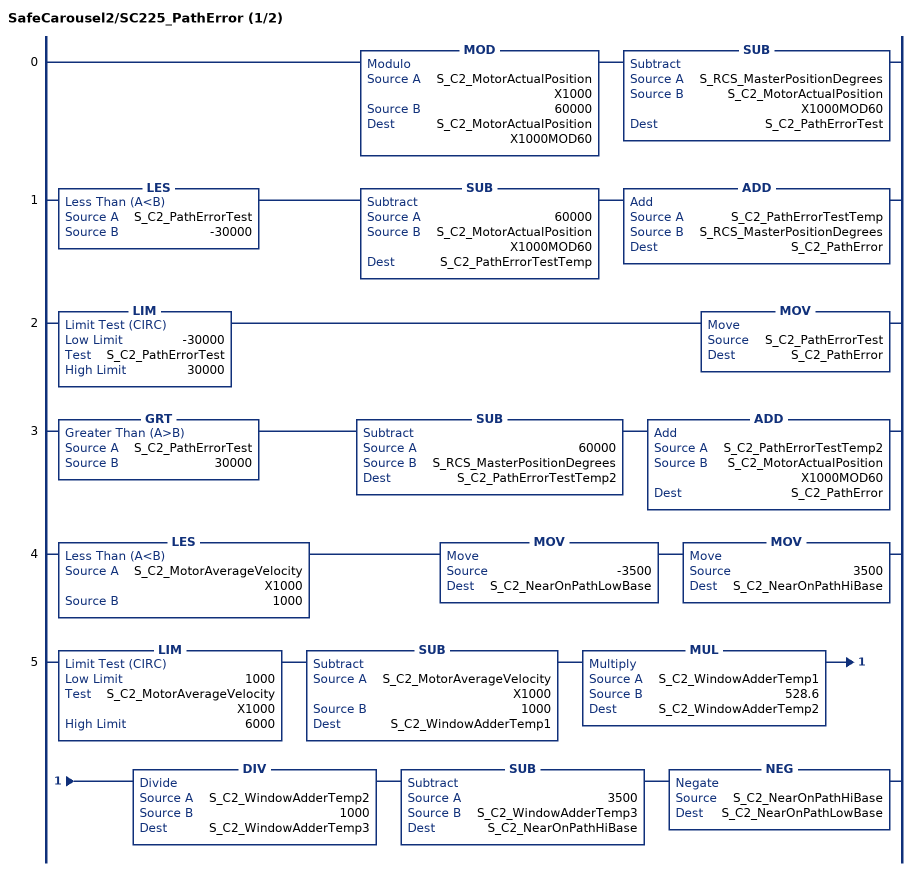
   0: MOD(S_C2_MotorActualPositionX1000,60000,S_C2_MotorActualPositionX1000MOD60)SUB(S_RCS_MasterPositionDegrees,S_C2_MotorActualPositionX1000MOD60,S_C2_PathErrorTest);
   1: LES(S_C2_PathErrorTest,-30000)SUB(60000,S_C2_MotorActualPositionX1000MOD60,S_C2_PathErrorTestTemp)ADD(S_C2_PathErrorTestTemp,S_RCS_MasterPositionDegrees,S_C2_PathError);
   2: LIM(-30000,S_C2_PathErrorTest,30000)MOV(S_C2_PathErrorTest,S_C2_PathError);
   3: GRT(S_C2_PathErrorTest,30000)SUB(60000,S_RCS_MasterPositionDegrees,S_C2_PathErrorTestTemp2)ADD(S_C2_PathErrorTestTemp2,S_C2_MotorActualPositionX1000MOD60,S_C2_PathError);
   4: LES(S_C2_MotorAverageVelocityX1000,1000)MOV(-3500,S_C2_NearOnPathLowBase)MOV(3500,S_C2_NearOnPathHiBase);
   5: LIM(1000,S_C2_MotorAverageVelocityX1000,6000)SUB(S_C2_MotorAverageVelocityX1000,1000,S_C2_WindowAdderTemp1)MUL(S_C2_WindowAdderTemp1,528.6,S_C2_WindowAdderTemp2)DIV(S_C2_WindowAdderTemp2,1000,S_C2_WindowAdderTemp3)SUB(3500,S_C2_WindowAdderTemp3,S_C2_NearOnPathHiBase)NEG(S_C2_NearOnPathHiBase,S_C2_NearOnPathLowBase);
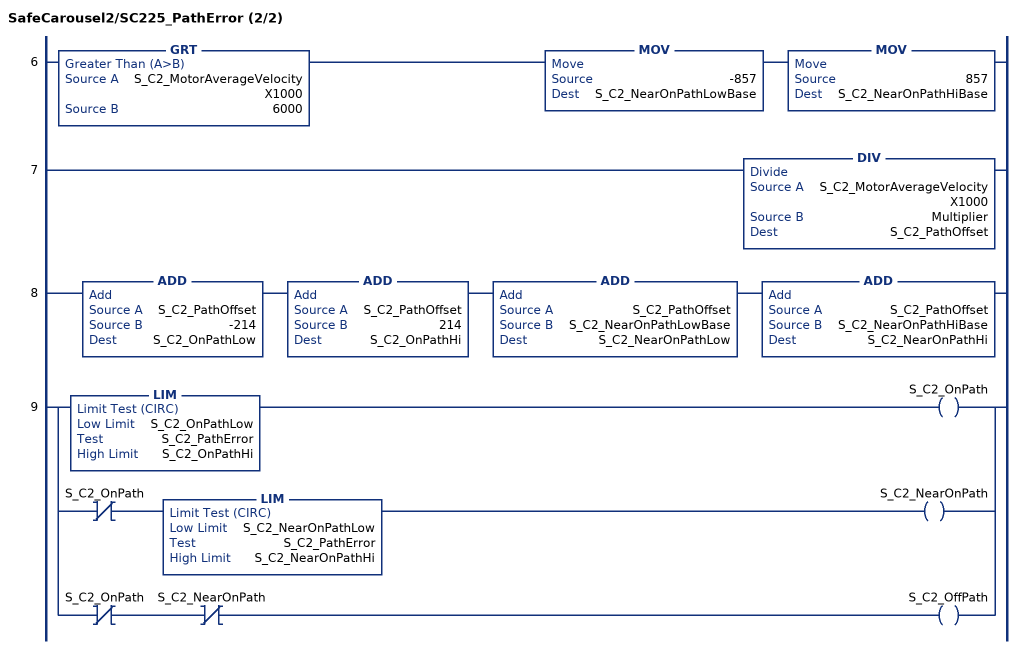
   6: GRT(S_C2_MotorAverageVelocityX1000,6000)MOV(-857,S_C2_NearOnPathLowBase)MOV(857,S_C2_NearOnPathHiBase);
   7: DIV(S_C2_MotorAverageVelocityX1000,Multiplier,S_C2_PathOffset);
   8: ADD(S_C2_PathOffset,-214,S_C2_OnPathLow)ADD(S_C2_PathOffset,214,S_C2_OnPathHi)ADD(S_C2_PathOffset,S_C2_NearOnPathLowBase,S_C2_NearOnPathLow)ADD(S_C2_PathOffset,S_C2_NearOnPathHiBase,S_C2_NearOnPathHi);
   9: [LIM(S_C2_OnPathLow,S_C2_PathError,S_C2_OnPathHi) OTE(S_C2_OnPath) ,XIO(S_C2_OnPath) LIM(S_C2_NearOnPathLow,S_C2_PathError,S_C2_NearOnPathHi) OTE(S_C2_NearOnPath) ,XIO(S_C2_OnPath) XIO(S_C2_NearOnPath) OTE(S_C2_OffPath) ];
END_ROUTINE
